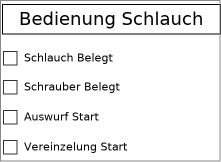
VISUALIZATION Frame_Schlauch_Bedien  // 221x162
VAR_IN_OUT
	bSchlauchBelegt			:BOOL;
	bSchrauberBelegt		:BOOL;
	bAuswurfStart			:BOOL;
	bVereinzelungStart		:BOOL;
END_VAR
    Checkbox (1,72 150x30), "Schrauber Belegt", variable: bSchrauberBelegt
    Checkbox (1,43 150x30), "Schlauch Belegt", variable: bSchlauchBelegt
    Checkbox (1,102 150x30), "Auswurf Start", variable: bAuswurfStart
    Checkbox (1,132 150x30), "Vereinzelung Start", variable: bVereinzelungStart
    Rectangle (2,4 219x30), "Bedienung Schlauch"
END_VISUALIZATION

(* stored: Version 1.1.0.1, ProductVersion 3.1.4024.15
   Visu Frame_Schlauch_Bedien: Id {cd3ad232-f842-4e20-9d8a-91ae491ee4ef} *)
